Staubli VAL3: ReadAction.pgx

public program ReadAction(bool& x_bRes (dimensions=1))
  local num l_nNum[3]
  local string l_sBuff
  local string l_sFileName
begin

  //读取动作文本
  //动作一共是200项，每项12个动作，每个动作一共是一个值
  //


  //参数初始化
  x_bRes=false
  l_sFileName="Disk://Txt/Action.txt"

  //判断文件是否存在
  if !$fileExists(l_sFileName)
    return
  endIf

  //关闭所有文件
  call FileDir:CloseAllFile()

  //文件是否可以打开
  nFileID=$fileOpen(l_sFileName,"r")
  if nFileID<0 or nFileID>9
    return
  endIf

  //对于原有值进行初始化
  for l_nNum[0]=0 to 50
    for l_nNum[1]=0 to 11
      for l_nNum[2]=0 to 1
        nAction[l_nNum[0],l_nNum[1],l_nNum[2]]=0
      endFor
    endFor
  endFor

  l_nNum[0]=l_nNum[1]=l_nNum[2]=0


  //读取每行并解析
  while $fileGet(nFileID,l_sBuff,1)==1 and l_sBuff!="" and l_nNum[0]<51
    call FileDir:SplitActionLine(l_sBuff,nAction,l_nNum[0]+1,x_bRes)
    if !x_bRes
      return
    endIf
    l_nNum[0]=l_nNum[0]+1
  endWhile
  //关闭所有文件
  call FileDir:CloseAllFile()
  x_bRes=true

end
